// TIA Portal project "FB ESTRELLA-TRIANGULO" (V11)

(* hardware
DEVICE "S7300/ET200 station_1"  SIMATIC 300-Station
   slot 0: "Perfil soporte_0"  Rail  6ES7 390-1***0-0AA0
   slot 1: "PS 307 2A_1"  PS 307 2A  6ES7 307-1BA00-0AA0
   slot 2: "PLC_1"  CPU 313C-2 DP  6ES7 313-6CF03-0AB0  V2.6
      slot 0: "Interfaz MPI_1"  MPI
      slot 1: "Interfaz DP_1"  DP
      slot 2: "DI16/DO16_1"  DI16/DO16
      slot 4: "Contaje_1"  Counter
   slot 4: "AI4/AO2 x 8bits_1"  AI4/AO2x8/8Bit  6ES7 334-0CE01-0AA0
   slot 5: "CP 343-1 Lean_1"  CP 343-1 LEAN  6GK7 343-1CX10-0XE0  V2.4
   slot 6: "CP 340 RS232C_1"  CP 340 RS232C  6ES7 340-1AH02-0AE0  V1.0
   slot 7: "CP 340 RS422/485_1"  CP 340 RS422/485  6ES7 340-1CH02-0AE0  V1.0
*)

// ===== PLC "PLC_1"  CPU 313C-2 DP =====

VAR_GLOBAL   // PLC tag table "Tabla de variables estándar"
   "MARCHA" AT %E0.0 : Bool;
   "PARO" AT %E0.1 : Bool;
   "LINEA" AT %A0.0 : Bool;
   "Tag_1" AT %T0 : Timer;
   "ESTRELLA" AT %A0.1 : Bool;
   "TRIANGULO" AT %A0.2 : Bool;
   "Tag_2" AT %T1 : Timer;
   "Tag_3" AT %I0.2 : Bool;
   "Tag_4" AT %I0.3 : Bool;
   "Tag_5" AT %Q0.3 : Bool;
   "Tag_6" AT %T2 : Timer;
END_VAR

DATA_BLOCK "ESTRELLA -TRIANGULO_DB_2"   // DB3
{ S7_Optimized_Access := 'FALSE' }
VERSION : 0.1
// stored: InstanceOfName ESTRELLA -TRIANGULO
"ESTRELLA -TRIANGULO"
BEGIN
END_DATA_BLOCK

FUNCTION_BLOCK "ESTRELLA -TRIANGULO"   // FB1, LAD
{ S7_Optimized_Access := 'FALSE' }
VERSION : 0.1
   VAR_INPUT
      MARCHA : Bool;
      PARO : Bool;
      TEMPORIZADOR : Timer;
      TIEMPO : S5Time;
   END_VAR
   VAR_OUTPUT
      LINEA : Bool;
      ESTRELLA : Bool;
      TRIANGULO : Bool;
   END_VAR
   VAR
      B0 : Bool;
      B1 : Bool;
      B2 : Bool;
      B3 : Bool;
      F4 : Bool;
      F5 : Bool;
      F6 : Bool;
      F7 : Bool;
   END_VAR
BEGIN

REGION Network 1
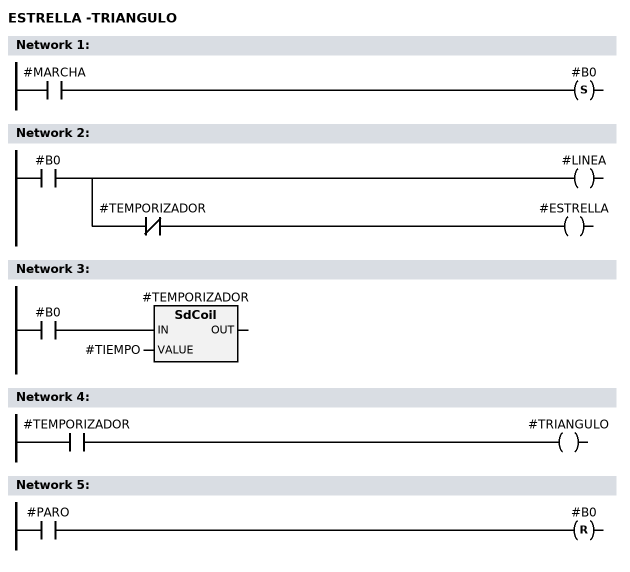
   RUNG wire#powerrail
      Contact( #MARCHA )
      S_Coil( #B0 )
   END_RUNG
   // the same network as SCL:
   IF #MARCHA THEN #B0 := TRUE; END_IF;
END_REGION

REGION Network 2
   RUNG wire#powerrail
      Contact( #B0 )
      wire#w1
      Coil( #LINEA )
   END_RUNG
   RUNG wire#w1
      I_Contact( #TEMPORIZADOR )
      Coil( #ESTRELLA )
   END_RUNG
   // the same network as SCL:
   #LINEA := #B0;
   #ESTRELLA := #B0 AND NOT #TEMPORIZADOR;
END_REGION

REGION Network 3
   // no SCL statement known for SdCoil: written as a call
   SdCoil(in := #B0, value := #TIEMPO, operand := #TEMPORIZADOR);
END_REGION

REGION Network 4
   RUNG wire#powerrail
      Contact( #TEMPORIZADOR )
      Coil( #TRIANGULO )
   END_RUNG
   // the same network as SCL:
   #TRIANGULO := #TEMPORIZADOR;
END_REGION

REGION Network 5
   RUNG wire#powerrail
      Contact( #PARO )
      R_Coil( #B0 )
   END_RUNG
   // the same network as SCL:
   IF #PARO THEN #B0 := FALSE; END_IF;
END_REGION
END_FUNCTION_BLOCK

ORGANIZATION_BLOCK "Main"   // OB1, LAD
TITLE = "Main Program Sweep (Cycle)"
{ S7_Optimized_Access := 'FALSE' }
VERSION : 0.1
   VAR_TEMP
      OB1_EV_CLASS : Byte;   // Bits 0-3 = 1 (Coming event), Bits 4-7 = 1 (Event class 1)
      OB1_SCAN_1 : Byte;   // 1 (Cold restart scan 1 of OB 1), 3 (Scan 2-n of OB 1)
      OB1_PRIORITY : Byte;   // Priority of OB Execution
      OB1_OB_NUMBR : Byte;   // 1 (Organization block 1, OB1)
      OB1_RESERVED_1 : Byte;   // Reserved for system
      OB1_RESERVED_2 : Byte;   // Reserved for system
      OB1_PREV_CYCLE : Int;   // Cycle time of previous OB1 scan (milliseconds)
      OB1_MIN_CYCLE : Int;   // Minimum cycle time of OB1 (milliseconds)
      OB1_MAX_CYCLE : Int;   // Maximum cycle time of OB1 (milliseconds)
      OB1_DATE_TIME : Date_And_Time;   // Date and time OB1 started
   END_VAR
BEGIN

REGION Network 1
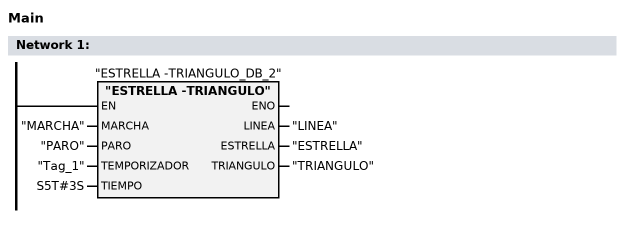
   RUNG wire#powerrail
      "ESTRELLA -TRIANGULO_DB_2"(MARCHA := "MARCHA", PARO := "PARO", TEMPORIZADOR := "Tag_1", TIEMPO := S5T#3S, LINEA => "LINEA", ESTRELLA => "ESTRELLA", TRIANGULO => "TRIANGULO")
   END_RUNG
   // the same network as SCL:
   "ESTRELLA -TRIANGULO_DB_2"(MARCHA := "MARCHA",   // "ESTRELLA -TRIANGULO"
                           PARO := "PARO",
                           TEMPORIZADOR := "Tag_1",
                           TIEMPO := S5T#3S,
                           LINEA => "LINEA",
                           ESTRELLA => "ESTRELLA",
                           TRIANGULO => "TRIANGULO");
END_REGION
END_ORGANIZATION_BLOCK